// TIA Portal V17 export
// export: Created 2024-08-26T21:07:21.6265614Z, ExportSetting WithDefaults, DisplayName Totally Integrated Automation Portal, DisplayVersion V17 Update 7, DisplayName TIA Portal Openness, DisplayVersion V17 Update 7, DisplayName TIA Portal Version Control Interface, DisplayVersion V17, DisplayName SINAMICS Startdrive Advanced, DisplayVersion V17 SP2, DisplayName SINAMICS Startdrive G110M, G120, G120C, G120D, G120P, G115D, DisplayVersion V17 SP2, DisplayName SINAMICS Startdrive G130, G150, S120, S150, SINAMICS MV, S210, DisplayVersion V17 SP2, DisplayName STEP 7 Professional, DisplayVersion V17 Update 7, DisplayName STEP 7 Safety, DisplayVersion V17 Update 6, DisplayName WinCC Advanced / Unified PC, DisplayVersion V17 Update 7
VAR_GLOBAL   // PLC tag table "digitalFieldbusInputs"
   iRightManualRodInsExt AT %I156.5 : Bool;
   iLeftToolingLockExt AT %I1.3 : Bool;
   iRightToolingExt AT %I156.7 : Bool;
   iTorqueToolingExt AT %I156.6 : Bool;
   iRigthManualRodInsRet AT %I157.5 : Bool;
   iLeftToolingLockRet AT %I1.4 : Bool;
   iRightToolingRet AT %I157.7 : Bool;
   iTorqueToolingRet AT %I157.6 : Bool;
   iStrapDetection AT %I45.3 : Bool;
   iLeftBracketDetection AT %I45.2 : Bool;
   iPresLeftManFrame AT %I157.1 : Bool;
   iRightBracketDetection AT %I45.0 : Bool;
   iManualExtOk AT %I158.3 : Bool;
   iProductInsertedLh AT %I45.1 : Bool;
   iLeftHomePos AT %I159.6 : Bool;
   iLeftWorkPos AT %I158.6 : Bool;
   iLeftToolingPos3 AT %I158.7 : Bool;
   iManualExtNok AT %I159.3 : Bool;
   iPresRightPwrFrame AT %I156.3 : Bool;
   iManualBumper AT %I158.5 : Bool;
   iLeftSpringColor AT %I158.2 : Bool;
   iRightSpringColor AT %I158.4 : Bool;
   iLeftManualRodInsRet AT %I157.4 : Bool;
   iInsertionCylindersRet AT %I1.2 : Bool;
   iInsertionCylindersExt AT %I1.1 : Bool;
   iLeftManToolingExtNok AT %I159.7 : Bool;
   iProductInsertedRh AT %I45.6 : Bool;
   iTorqueToolingHome AT %I45.5 : Bool;
   iRightToolinPos1 AT %I156.4 : Bool;
   iRightToolinPos3 AT %I156.2 : Bool;
   iRightToolinPos2 AT %I157.2 : Bool;
   iManualZExtOk AT %I156.0 : Bool;
   iManualZExtNok AT %I157.0 : Bool;
   iRightManToolingRet AT %I158.1 : Bool;
   iTorqueTrigger AT %I160.0 : Bool;
   toolingID1 AT %I1.5 : Bool;
   manualProductPres AT %Q10.0 : Bool;
   powerProductPres AT %Q10.1 : Bool;
END_VAR
